{region '#Template'}
	{attribute 'Version' := '5.0.0.0'}
	{attribute 'Tags' := '"LCID": "1031", "Text": "Trade, Plant, General"'}
	{attribute 'Tags' := '"LCID": "1033", "Text": "Trade, Plant, General"'}
	{attribute 'Using' := '"Type": "Template", "URI": "Site"'}
	{attribute 'Description' := '"LCID": "1031", "Text": "Aufruf der Anlagen des Gewerks Allgemein"'}
	{attribute 'Description' := '"LCID": "1033", "Text": "Calling the plants of the trade general"'}
{endregion}
FUNCTION_BLOCK FB_BA_BuildingAutomation EXTENDS FB_BA_View
VAR_INPUT
END_VAR
VAR_INPUT CONSTANT
	BuildingGlobal		: FB_BA_EventsAndSettings;
	Weatherstation		: FB_BA_WeatherStation_Draft;			
	AdsComServer		: FB_BA_AdsComServer;	
	//AdsComClient		: FB_BA_AdsComClient;	
END_VAR

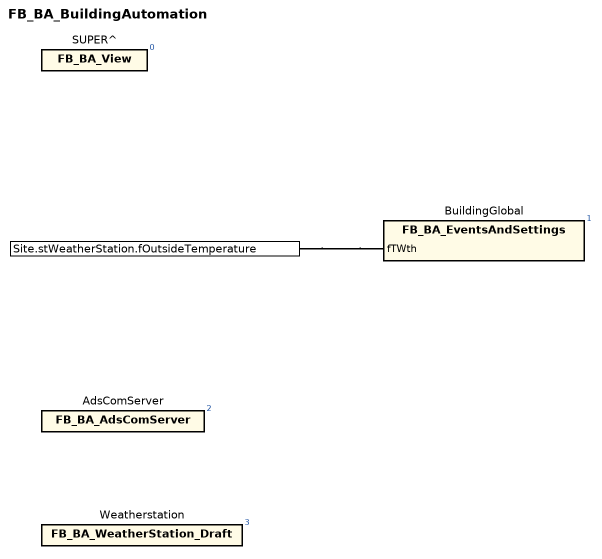
SUPER^(); // FB_BA_View
BuildingGlobal(fTWth := Site.stWeatherStation.fOutsideTemperature); // FB_BA_EventsAndSettings
AdsComServer(); // FB_BA_AdsComServer
Weatherstation(); // FB_BA_WeatherStation_Draft

METHOD FB_init : BOOL
VAR_INPUT
	bInitRetains : BOOL; // if TRUE, the retain variables are initialized (warm start / cold start)
	bInCopyCode : BOOL;  // if TRUE, the instance afterwards gets moved into the copy code (online change)
END_VAR
								


				 
BuildingGlobal.iParent			:= THIS^;	
BuildingGlobal.iLabel			:= LblPlt_Global_Building_Data;
BuildingGlobal.sObjectName		:= '{Idx=01}';
BuildingGlobal.eDPADMode		:= E_BA_DPADMode.eInclude;

//AdsComClient.iParent			:= THIS^;
//AdsComClient					:= LblPlt_Global_Building_Data;
//AdsComClient.sObjectName		:= '{Idx=02}';  
//AdsComClient.eDPADMode		:= E_BA_DPADMode.eInclude;

Weatherstation.iParent			:= THIS^;
Weatherstation.iLabel			:= LblPlt_Weather_station;
Weatherstation.sObjectName		:= '{Idx=01}';
Weatherstation.eDPADMode		:= E_BA_DPADMode.eInclude;
END_METHOD

END_FUNCTION_BLOCK

(* stored: Version 1.1.0.1, ProductVersion 3.1.4024.12
   POU FB_BA_BuildingAutomation: Id {37715593-93b1-401c-b83d-b5a4c7d7c41e}, SpecialFunc None
   Method FB_init: Id {63ef2833-b0ed-49d1-b83a-d3b3ee61d402} *)
